Staubli VAL3: onF7Event.pgx

program onF7Event()
  local string l_sMessage
  local bool l_bContinue
  local string l_sProgram
  local num l_nZero
begin
  // look if the bButton is enable
  if bButton[6]
    //
    // STOP/START CYCLE
    //
    if cycleStatus:bCycle
      logMsg("[KERNEL] INTERFACE:Stop cycle")
      stopMove()
      cycleStatus:bToStop=true
      call use:timerDialog(" STOP CYCLE ",1)
      watch(cycleStatus:bToStop==false,1)
    else
      // start cycle
      l_nZero=0
      call processList:getCycle(l_sProgram,l_nZero,l_nZero,l_nZero,1)
      if l_sProgram!=""
        //if (cycleStatus:nWorkingMode==3 or cycleStatus:nWorkingMode==4)
        logMsg("[KERNEL] INTERFACE:Start cycle")
        cycleStatus:bToStart=true
        wait(cycleStatus:bToStart==false)
      else
        // program in the process List
        call language:message(l_sMessage,91)
        popUpMsg(l_sMessage)
      endIf
    endIf
    call use:nullKey(nKey)
  endIf
end
